TYPE state :
(
	INIT,
	POWER_ON,
	MOVE_ON,
	ERROR,
	P_RESET
)UDINT;
END_TYPE

(* stored: Version 1.1.0.1, ProductVersion 3.1.4024.9
   DUT state: Id {85b9a111-64c9-4594-81d3-778cc125adb4} *)
